% RSLogix 500 project Q6.RSS, saved by version 8.30.00.16 %
PROJECT "Q6"    % processor: Bul.1763 MicroLogix 1100 Series B %

PROGRAM FILES
  LAD 2   8 rungs

DATA FILES
  O0 OUTPUT  4 elements
  I1 INPUT  6 elements
  S2 STATUS  66 elements
  B3 BINARY  1 elements
  T4 TIMER  3 elements
  C5 COUNTER  1 elements
  R6 CONTROL  1 elements
  N7 INTEGER  1 elements
  F8 FLOAT  1 elements

LADDER 2
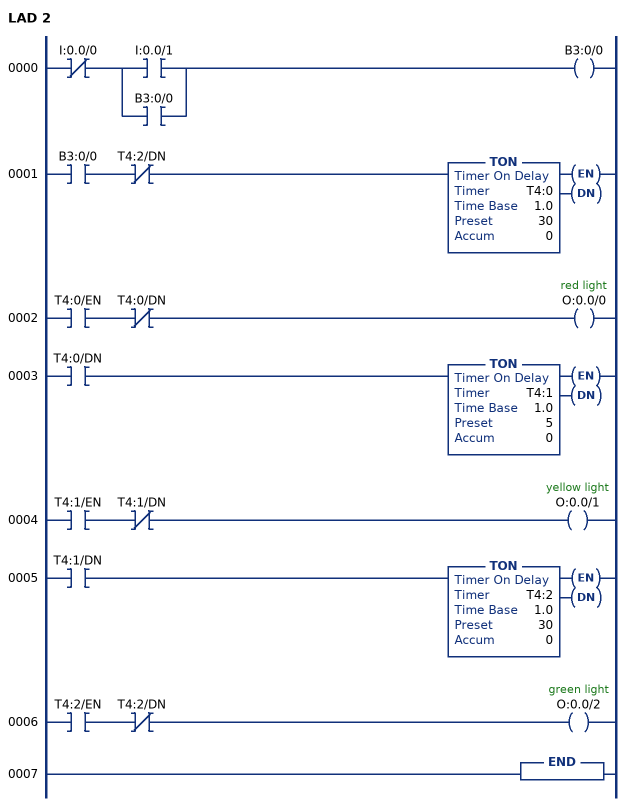
% Rung: 0 %
SOR XIO I:0.0/0 BST XIC I:0.0/1 NXB XIC B3:0/0 BND OTE B3:0/0 EOR
% Rung: 1 %
SOR XIC B3:0/0 XIO T4:2/DN TON T4:0 1.0 30 0 EOR
% Rung: 2 %
SOR XIC T4:0/EN XIO T4:0/DN OTE O:0.0/0 EOR
%   O:0.0/0  "red light" %
% Rung: 3 %
SOR XIC T4:0/DN TON T4:1 1.0 5 0 EOR
% Rung: 4 %
SOR XIC T4:1/EN XIO T4:1/DN OTE O:0.0/1 EOR
%   O:0.0/1  "yellow light" %
% Rung: 5 %
SOR XIC T4:1/DN TON T4:2 1.0 30 0 EOR
% Rung: 6 %
SOR XIC T4:2/EN XIO T4:2/DN OTE O:0.0/2 EOR
%   O:0.0/2  "green light" %
% Rung: 7 %
SOR END EOR

DATA TABLE (non-zero values as saved)
DATA T4
% .PRE .ACC %
% T4:0 % 30 0
% T4:1 % 5 0
% T4:2 % 30 0
